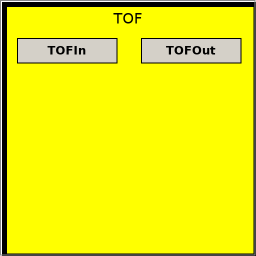
VISUALIZATION V_PH_TOF  // 256x256
VAR_INPUT
	stSafetyTOF			:ST_SAFETY_FBTOF;
END_VAR
    Rectangle (2,2 256x256), colour toggle: stSafetyTOF.bGeneralError
    Label (5,6 246x25), "TOF"
    RoundedRectangle (17,38 100x25), "TOFIn", colour toggle: stSafetyTOF.uStatus.stStatusWords.wInputs.8
    RoundedRectangle (141,38 100x25), "TOFOut", colour toggle: stSafetyTOF.uStatus.stStatusWords.wOutputs.1
    Textfield (17,226 234x25), text list: 'TL_FbStateTimer', text index: stSafetyTOF.eState
END_VISUALIZATION

(* stored: Version 1.1.0.1, ProductVersion 3.1.4024.4
   Visu V_PH_TOF: Id {2d26c9b5-e5ec-46a3-8223-6187b7e5fdaf} *)
